// TIA Portal project "自动组装流水线（核心程序）" (V16)

(* hardware
DEVICE "S7-1200 station_1"  S7-1200 Station
   slot 0: "Rack_0"  S7-1200 Rack  Rack  V1.0
   slot 1: "PLC_1"  CPU 1214C DC/DC/Rly  6ES7 214-1HG40-0XB0  V4.4
*)

// ===== PLC "PLC_1"  CPU 1214C DC/DC/Rly =====

VAR_GLOBAL   // PLC tag table "io"
   "传感器9" AT %I0.0 : Bool;
   "传感器8" AT %I0.1 : Bool;
   "传感器7" AT %I0.2 : Bool;
   "传感器1" AT %I0.3 : Bool;
   "传感器2" AT %I0.4 : Bool;
   "传感器3" AT %I0.5 : Bool;
   "传感器4" AT %I0.6 : Bool;
   "传感器5" AT %I0.7 : Bool;
   "传感器6" AT %I1.0 : Bool;
   "传感器10" AT %I1.1 : Bool;
   "开始" AT %I1.2 : Bool;
   "复位" AT %I1.3 : Bool;
   "停止" AT %I1.4 : Bool;
   "紧急停止" AT %I1.5 : Bool;
   "1挡" AT %I1.6 : Bool;
   "FACTORY I/O (Running)" AT %I1.7 : Bool;
   "前后" AT %Q0.0 : Bool;
   "上下" AT %Q0.1 : Bool;
   "吸取" AT %Q0.2 : Bool;
   "皮带1" AT %Q0.3 : Bool;
   "推上盖" AT %Q0.4 : Bool;
   "上升1" AT %Q0.5 : Bool;
   "皮带2" AT %Q0.6 : Bool;
   "推下盖" AT %Q0.7 : Bool;
   "上升2" AT %Q1.0 : Bool;
   "绿灯" AT %Q1.1 : Bool;
   "黄灯" AT %Q1.2 : Bool;
   "红灯" AT %Q1.3 : Bool;
   "显示屏" AT %QD30 : DInt;
END_VAR

VAR_GLOBAL   // PLC tag table "中间变量"
   "中间变量1" AT %M0.0 : Bool;
   "中间变量2" AT %M0.1 : Bool;
   "中间变量3" AT %M0.2 : Bool;
   "中间变量4" AT %M0.3 : Bool;
   "中间变量5" AT %M0.4 : Bool;
   "中间变量6" AT %M0.5 : Bool;
   "中间变量7" AT %M0.6 : Bool;
   "中间变量8" AT %M0.7 : Bool;
   "中间变量9" AT %M1.0 : Bool;
   "中间变量10" AT %M1.1 : Bool;
   "中间变量11" AT %M1.2 : Bool;
   "中间变量12" AT %M1.3 : Bool;
   "中间变量13" AT %M1.4 : Bool;
   "中间变量14" AT %M1.5 : Bool;
   "启动" AT %M1.6 : Bool;
   "停止(1)" AT %M1.7 : Bool;
   "复位(1)" AT %M2.0 : Bool;
   "启动标志1" AT %M2.1 : Bool;
   "推杆标志1" AT %M2.2 : Bool;
   "推杆标志2" AT %M2.3 : Bool;
   "推杆收1" AT %M2.4 : Bool;
   "推杆收2" AT %M2.5 : Bool;
   "上下准备" AT %M2.6 : Bool;
   "吸附准备" AT %M2.7 : Bool;
   "吸附过程" AT %M3.0 : Bool;
   "前后准备" AT %M3.1 : Bool;
   "准备下降" AT %M3.2 : Bool;
   "断开吸附" AT %M3.3 : Bool;
   "x轴复位" AT %M3.4 : Bool;
   "皮带1状态" AT %M3.5 : Bool;
   "皮带2状态" AT %M3.6 : Bool;
   "皮带启动1" AT %M3.7 : Bool;
   "皮带启动2" AT %M4.0 : Bool;
   "上升2准备" AT %M4.1 : Bool;
   "上升2复位" AT %M4.2 : Bool;
END_VAR

// folder: System blocks/Program resources

DATA_BLOCK "IEC_Timer_0_DB"   // DB1
{ S7_Optimized_Access := 'TRUE' }
AUTHOR : Simatic
FAMILY : IEC
NAME : IEC_TMR
VERSION : 1.0
// stored: InstanceOfName IEC_TIMER
"IEC_TIMER"
BEGIN
END_DATA_BLOCK

DATA_BLOCK "IEC_Timer_0_DB_1"   // DB2
{ S7_Optimized_Access := 'TRUE' }
AUTHOR : Simatic
FAMILY : IEC
NAME : IEC_TMR
VERSION : 1.0
// stored: InstanceOfName IEC_TIMER
"IEC_TIMER"
BEGIN
END_DATA_BLOCK

DATA_BLOCK "IEC_Timer_0_DB_2"   // DB3
{ S7_Optimized_Access := 'TRUE' }
AUTHOR : Simatic
FAMILY : IEC
NAME : IEC_TMR
VERSION : 1.0
// stored: InstanceOfName IEC_TIMER
"IEC_TIMER"
BEGIN
END_DATA_BLOCK

DATA_BLOCK "IEC_Timer_0_DB_3"   // DB4
{ S7_Optimized_Access := 'TRUE' }
AUTHOR : Simatic
FAMILY : IEC
NAME : IEC_TMR
VERSION : 1.0
// stored: InstanceOfName IEC_TIMER
"IEC_TIMER"
BEGIN
END_DATA_BLOCK

DATA_BLOCK "IEC_Timer_0_DB_4"   // DB5
{ S7_Optimized_Access := 'TRUE' }
AUTHOR : Simatic
FAMILY : IEC
NAME : IEC_TMR
VERSION : 1.0
// stored: InstanceOfName IEC_TIMER
"IEC_TIMER"
BEGIN
END_DATA_BLOCK

DATA_BLOCK "IEC_Timer_0_DB_5"   // DB6
{ S7_Optimized_Access := 'TRUE' }
AUTHOR : Simatic
FAMILY : IEC
NAME : IEC_TMR
VERSION : 1.0
// stored: InstanceOfName IEC_TIMER
"IEC_TIMER"
BEGIN
END_DATA_BLOCK

DATA_BLOCK "IEC_Timer_0_DB_6"   // DB7
{ S7_Optimized_Access := 'TRUE' }
AUTHOR : Simatic
FAMILY : IEC
NAME : IEC_TMR
VERSION : 1.0
// stored: InstanceOfName IEC_TIMER
"IEC_TIMER"
BEGIN
END_DATA_BLOCK

DATA_BLOCK "IEC_Timer_0_DB_7"   // DB8
{ S7_Optimized_Access := 'TRUE' }
AUTHOR : Simatic
FAMILY : IEC
NAME : IEC_TMR
VERSION : 1.0
// stored: InstanceOfName IEC_TIMER
"IEC_TIMER"
BEGIN
END_DATA_BLOCK

DATA_BLOCK "IEC_Timer_0_DB_8"   // DB9
{ S7_Optimized_Access := 'TRUE' }
AUTHOR : Simatic
FAMILY : IEC
NAME : IEC_TMR
VERSION : 1.0
// stored: InstanceOfName IEC_TIMER
"IEC_TIMER"
BEGIN
END_DATA_BLOCK

DATA_BLOCK "IEC_Timer_0_DB_9"   // DB10
{ S7_Optimized_Access := 'TRUE' }
AUTHOR : Simatic
FAMILY : IEC
NAME : IEC_TMR
VERSION : 1.0
// stored: InstanceOfName IEC_TIMER
"IEC_TIMER"
BEGIN
END_DATA_BLOCK

DATA_BLOCK "IEC_Timer_0_DB_10"   // DB11
{ S7_Optimized_Access := 'TRUE' }
AUTHOR : Simatic
FAMILY : IEC
NAME : IEC_TMR
VERSION : 1.0
// stored: InstanceOfName IEC_TIMER
"IEC_TIMER"
BEGIN
END_DATA_BLOCK

DATA_BLOCK "IEC_Timer_0_DB_11"   // DB12
{ S7_Optimized_Access := 'TRUE' }
AUTHOR : Simatic
FAMILY : IEC
NAME : IEC_TMR
VERSION : 1.0
// stored: InstanceOfName IEC_TIMER
"IEC_TIMER"
BEGIN
END_DATA_BLOCK

// folder: (top level)

FUNCTION "MHJ-PLC-Lab-Function-S71200" : Void   // FC9000, SCL
{ S7_Optimized_Access := 'TRUE' }
VERSION : 0.1
   VAR_TEMP
      rdTimeReturn : Int;
      outputTime : DTL;
      SyncVal : Byte;
      forVal : Int;
      forVal_2 : Int;
      Value : Byte;
   END_VAR
   VAR CONSTANT
      CompVal : Byte := 16#34;
      Value_01 : Byte := 16#11;
      Value_01_DW : DWord := 16#A165_D992;
      Value_02_DW : DWord := 16#58BE_4401;
   END_VAR
BEGIN

   #Value:=PEEK(area := 16#82,
        dbNumber := 0,
        byteOffset := 511);
   #Value := #Value + 1;

   POKE(area := 16#82,
        dbNumber := 0,
        byteOffset := 511,
        value := #Value);

   POKE(area:=16#81,
        dbNumber:=0,
        byteOffset:=1016,
        value:=#Value_01_DW);
   POKE(area := 16#81,
        dbNumber := 0,
        byteOffset := 1020,
        value := #Value_02_DW);

   POKE(area := 16#81,
        dbNumber := 0,
        byteOffset := 511,
        value := B#16#00);

   FOR #forVal := 0 TO 120 DO
       FOR #forVal_2:=0 TO 10 DO
           #rdTimeReturn:=RD_SYS_T(#outputTime);
           #rdTimeReturn := WR_SYS_T(#outputTime);
           #rdTimeReturn := RD_SYS_T(#outputTime);
           #rdTimeReturn := WR_SYS_T(#outputTime);
       END_FOR;
       #SyncVal:= PEEK(area := 16#81,
                      dbNumber := 0,
                      byteOffset := 511);
       IF #SyncVal = #CompVal THEN
          GOTO M_1;
       END_IF;
   END_FOR;
   RETURN;

   M_1:
   POKE(area := 16#81,
        dbNumber := 0,
        byteOffset := 511,
        value := B#16#0);
END_FUNCTION

ORGANIZATION_BLOCK "Main"   // OB1, LAD, ProgramCycle
TITLE = "Main Program Sweep (Cycle)"
{ S7_Optimized_Access := 'TRUE' }
VERSION : 0.1
   VAR_INPUT
      Initial_Call : Bool;   // Initial call of this OB
      Remanence : Bool;   // =True, if remanent data are available
   END_VAR
   VAR_TEMP   // added for the SCL form of the ladder/FBD networks
      _w1 : Bool;
      _w2 : Bool;
   END_VAR
BEGIN

REGION Network 1
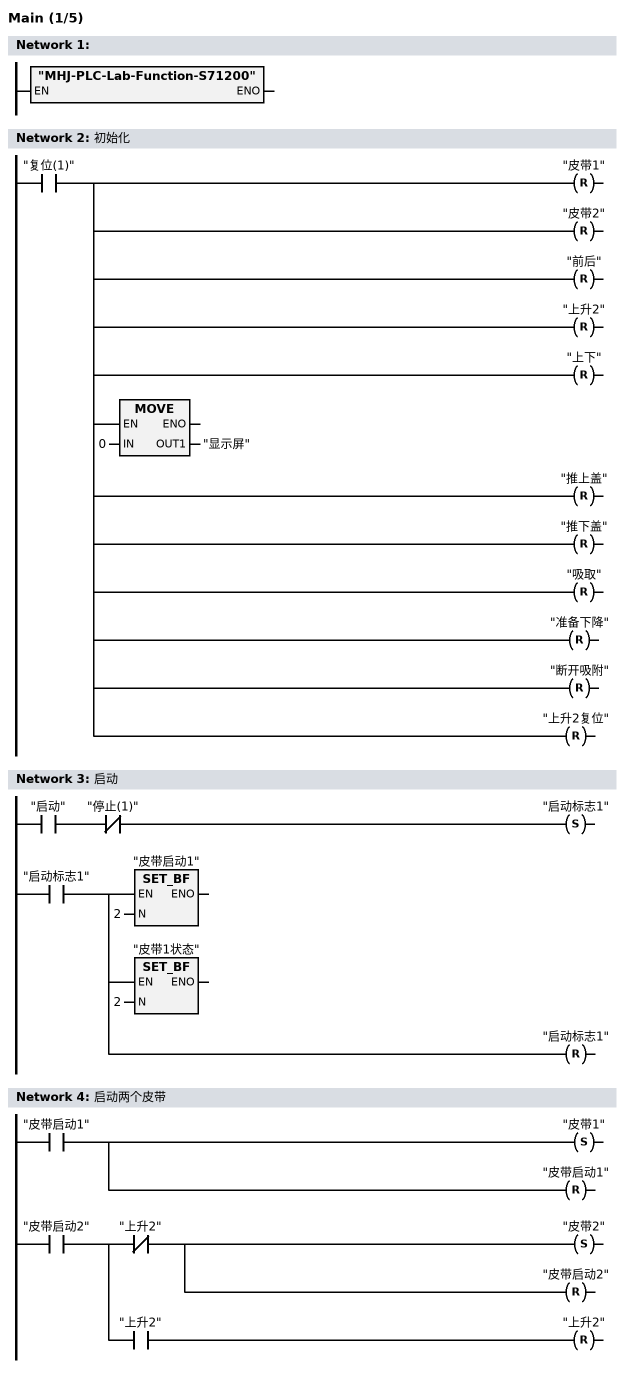
   RUNG wire#powerrail
      "MHJ-PLC-Lab-Function-S71200"()
   END_RUNG
   // the same network as SCL:
   "MHJ-PLC-Lab-Function-S71200"();
END_REGION

REGION Network 2: 初始化
   RUNG wire#powerrail
      Contact( "复位(1)" )
      wire#w1
      R_Coil( "皮带1" )
   END_RUNG
   RUNG wire#w1
      R_Coil( "皮带2" )
   END_RUNG
   RUNG wire#w1
      R_Coil( "前后" )
   END_RUNG
   RUNG wire#w1
      R_Coil( "上升2" )
   END_RUNG
   RUNG wire#w1
      R_Coil( "上下" )
   END_RUNG
   RUNG wire#w1
      Move(in := 0, out1 => "显示屏")
   END_RUNG
   RUNG wire#w1
      R_Coil( "推上盖" )
   END_RUNG
   RUNG wire#w1
      R_Coil( "推下盖" )
   END_RUNG
   RUNG wire#w1
      R_Coil( "吸取" )
   END_RUNG
   RUNG wire#w1
      R_Coil( "准备下降" )
   END_RUNG
   RUNG wire#w1
      R_Coil( "断开吸附" )
   END_RUNG
   RUNG wire#w1
      R_Coil( "上升2复位" )
   END_RUNG
   // the same network as SCL:
   IF "复位(1)" THEN
       "皮带1" := FALSE;
       "皮带2" := FALSE;
       "前后" := FALSE;
       "上升2" := FALSE;
       "上下" := FALSE;
       "显示屏" := 0;
       "推上盖" := FALSE;
       "推下盖" := FALSE;
       "吸取" := FALSE;
       "准备下降" := FALSE;
       "断开吸附" := FALSE;
       "上升2复位" := FALSE;
   END_IF;
END_REGION

REGION Network 3: 启动
   // no SCL statement known for SBitfield: written as a call
   IF "启动" AND NOT "停止(1)" THEN "启动标志1" := TRUE; END_IF;
   #_w1 := "启动标志1";
   IF #_w1 THEN
       SET_BF(operand := "皮带启动1", n := 2);
       SET_BF(operand := "皮带1状态", n := 2);
       "启动标志1" := FALSE;
   END_IF;
END_REGION

REGION Network 4: 启动两个皮带
   RUNG wire#powerrail
      Contact( "皮带启动1" )
      wire#w1
      S_Coil( "皮带1" )
   END_RUNG
   RUNG wire#w1
      R_Coil( "皮带启动1" )
   END_RUNG
   RUNG wire#powerrail
      Contact( "皮带启动2" )
      wire#w2
      I_Contact( "上升2" )
      wire#w3
      S_Coil( "皮带2" )
   END_RUNG
   RUNG wire#w3
      R_Coil( "皮带启动2" )
   END_RUNG
   RUNG wire#w2
      Contact( "上升2" )
      R_Coil( "上升2" )
   END_RUNG
   // the same network as SCL:
   IF "皮带启动1" THEN
       "皮带1" := TRUE;
       "皮带启动1" := FALSE;
   END_IF;
   IF "皮带启动2" AND NOT "上升2" THEN "皮带2" := TRUE; END_IF;
   #_w1 := "皮带启动2";
   IF "皮带启动2" AND NOT "上升2" THEN "皮带启动2" := FALSE; END_IF;
   IF #_w1 AND "上升2" THEN "上升2" := FALSE; END_IF;
END_REGION

REGION Network 5: 停止传送带运动，启动两个推杆
   // 因为传感器从1变为0在显示上面有延迟的存在，在电脑内部的运行中没有，所以需要延时一段时间，再停止运行皮带，开始运行推杆
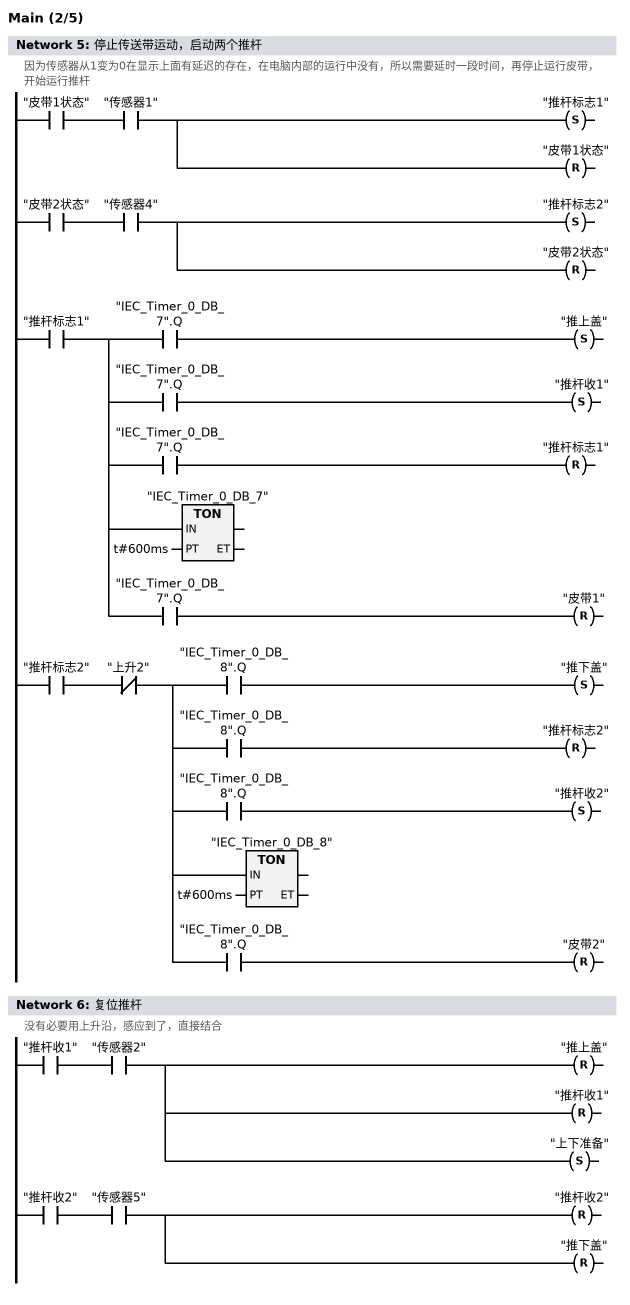
   IF "皮带1状态" AND "传感器1" THEN
       "推杆标志1" := TRUE;
       "皮带1状态" := FALSE;
   END_IF;
   IF "皮带2状态" AND "传感器4" THEN
       "推杆标志2" := TRUE;
       "皮带2状态" := FALSE;
   END_IF;
   IF "推杆标志1" AND "IEC_Timer_0_DB_7".Q THEN
       "推上盖" := TRUE;
       "推杆收1" := TRUE;
   END_IF;
   #_w1 := "推杆标志1";
   IF "推杆标志1" AND "IEC_Timer_0_DB_7".Q THEN "推杆标志1" := FALSE; END_IF;
   "IEC_Timer_0_DB_7".TON(IN := #_w1, PT := t#600ms);
   IF #_w1 AND "IEC_Timer_0_DB_7".Q THEN "皮带1" := FALSE; END_IF;
   #_w2 := "推杆标志2" AND NOT "上升2";
   IF #_w2 AND "IEC_Timer_0_DB_8".Q THEN
       "推下盖" := TRUE;
       "推杆标志2" := FALSE;
       "推杆收2" := TRUE;
   END_IF;
   "IEC_Timer_0_DB_8".TON(IN := #_w2, PT := t#600ms);
   IF #_w2 AND "IEC_Timer_0_DB_8".Q THEN "皮带2" := FALSE; END_IF;
END_REGION

REGION Network 6: 复位推杆
   // 没有必要用上升沿，感应到了，直接结合
   RUNG wire#powerrail
      Contact( "推杆收1" )
      Contact( "传感器2" )
      wire#w1
      R_Coil( "推上盖" )
   END_RUNG
   RUNG wire#w1
      R_Coil( "推杆收1" )
   END_RUNG
   RUNG wire#w1
      S_Coil( "上下准备" )
   END_RUNG
   RUNG wire#powerrail
      Contact( "推杆收2" )
      Contact( "传感器5" )
      wire#w2
      R_Coil( "推杆收2" )
   END_RUNG
   RUNG wire#w2
      R_Coil( "推下盖" )
   END_RUNG
   // the same network as SCL:
   IF "推杆收1" AND "传感器2" THEN "推上盖" := FALSE; END_IF;
   #_w1 := "推杆收1" AND "传感器2";
   IF #_w1 THEN
       "推杆收1" := FALSE;
       "上下准备" := TRUE;
   END_IF;
   #_w2 := "推杆收2" AND "传感器5";
   IF #_w2 THEN
       "推杆收2" := FALSE;
       "推下盖" := FALSE;
   END_IF;
END_REGION

REGION Network 7: 准备吸附
   // 利用传感器2来判断是否推到位
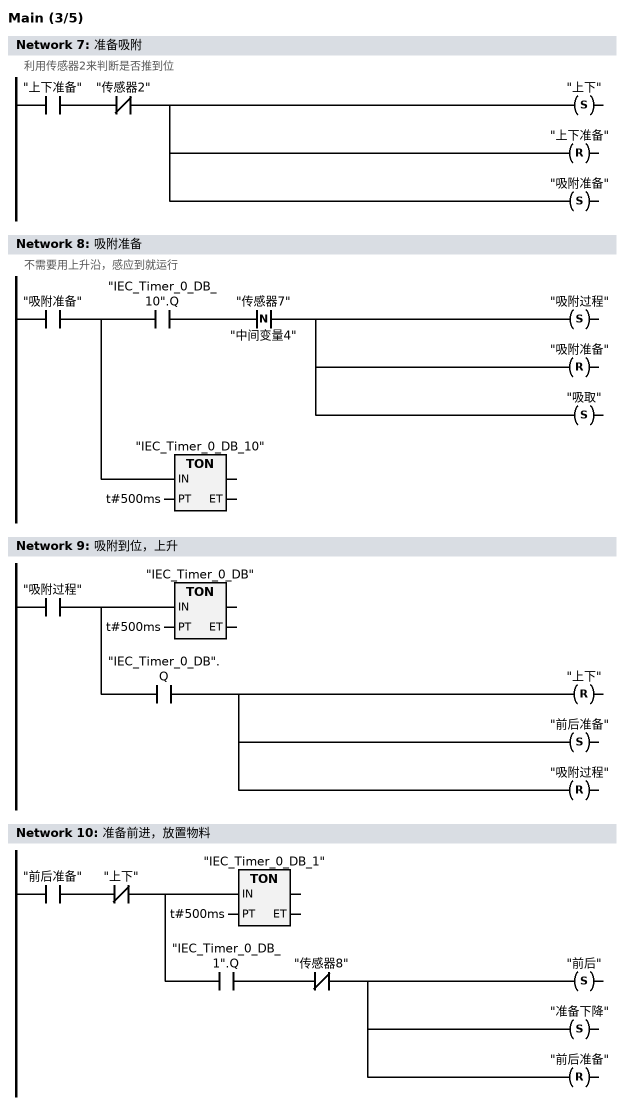
   RUNG wire#powerrail
      Contact( "上下准备" )
      I_Contact( "传感器2" )
      wire#w1
      S_Coil( "上下" )
   END_RUNG
   RUNG wire#w1
      R_Coil( "上下准备" )
   END_RUNG
   RUNG wire#w1
      S_Coil( "吸附准备" )
   END_RUNG
   // the same network as SCL:
   IF "上下准备" AND NOT "传感器2" THEN "上下" := TRUE; END_IF;
   #_w1 := "上下准备" AND NOT "传感器2";
   IF #_w1 THEN
       "上下准备" := FALSE;
       "吸附准备" := TRUE;
   END_IF;
END_REGION

REGION Network 8: 吸附准备
   // 不需要用上升沿，感应到就运行
   #_w1 := "吸附准备" AND "IEC_Timer_0_DB_10".Q AND NOT "传感器7" AND "中间变量4";   // falling edge of "传感器7"
   "中间变量4" := "传感器7";
   IF #_w1 THEN "吸附过程" := TRUE; END_IF;
   #_w2 := "吸附准备";
   IF #_w1 THEN
       "吸附准备" := FALSE;
       "吸取" := TRUE;
   END_IF;
   "IEC_Timer_0_DB_10".TON(IN := #_w2, PT := t#500ms);
END_REGION

REGION Network 9: 吸附到位，上升
   "IEC_Timer_0_DB".TON(IN := "吸附过程", PT := t#500ms);
   IF "吸附过程" AND "IEC_Timer_0_DB".Q THEN
       "上下" := FALSE;
       "前后准备" := TRUE;
       "吸附过程" := FALSE;
   END_IF;
END_REGION

REGION Network 10: 准备前进，放置物料
   #_w1 := "前后准备" AND NOT "上下";
   "IEC_Timer_0_DB_1".TON(IN := #_w1, PT := t#500ms);
   IF #_w1 AND "IEC_Timer_0_DB_1".Q AND NOT "传感器8" THEN
       "前后" := TRUE;
       "准备下降" := TRUE;
       "前后准备" := FALSE;
   END_IF;
END_REGION

REGION Network 11
   // 利用传感器不运动的时候，表示为0
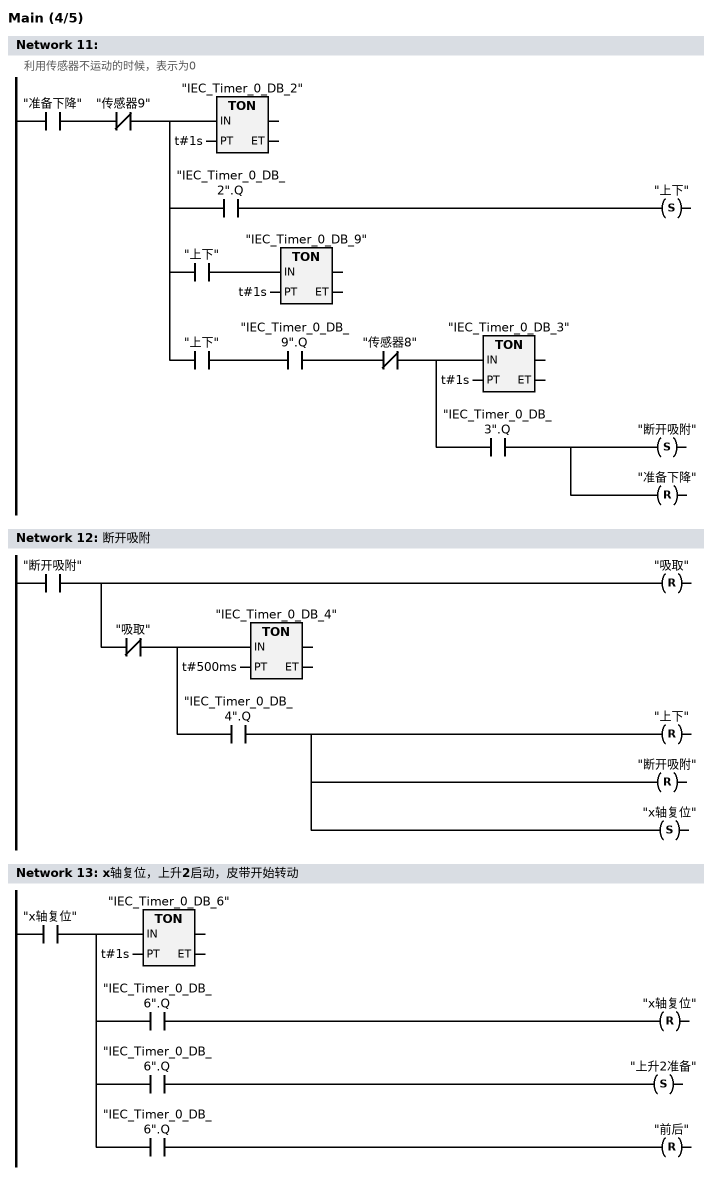
   #_w1 := "准备下降" AND NOT "传感器9";
   "IEC_Timer_0_DB_2".TON(IN := #_w1, PT := t#1s);
   IF #_w1 AND "IEC_Timer_0_DB_2".Q THEN "上下" := TRUE; END_IF;
   "IEC_Timer_0_DB_9".TON(IN := #_w1 AND "上下", PT := t#1s);
   #_w2 := #_w1 AND "上下" AND "IEC_Timer_0_DB_9".Q AND NOT "传感器8";
   "IEC_Timer_0_DB_3".TON(IN := #_w2, PT := t#1s);
   IF #_w2 AND "IEC_Timer_0_DB_3".Q THEN
       "断开吸附" := TRUE;
       "准备下降" := FALSE;
   END_IF;
END_REGION

REGION Network 12: 断开吸附
   IF "断开吸附" THEN "吸取" := FALSE; END_IF;
   #_w1 := "断开吸附" AND NOT "吸取";
   "IEC_Timer_0_DB_4".TON(IN := #_w1, PT := t#500ms);
   IF #_w1 AND "IEC_Timer_0_DB_4".Q THEN
       "上下" := FALSE;
       "断开吸附" := FALSE;
       "x轴复位" := TRUE;
   END_IF;
END_REGION

REGION Network 13: x轴复位，上升2启动，皮带开始转动
   "IEC_Timer_0_DB_6".TON(IN := "x轴复位", PT := t#1s);
   #_w1 := "x轴复位";
   IF "x轴复位" AND "IEC_Timer_0_DB_6".Q THEN "x轴复位" := FALSE; END_IF;
   IF #_w1 AND "IEC_Timer_0_DB_6".Q THEN
       "上升2准备" := TRUE;
       "前后" := FALSE;
   END_IF;
END_REGION

REGION Network 14: 准备循环
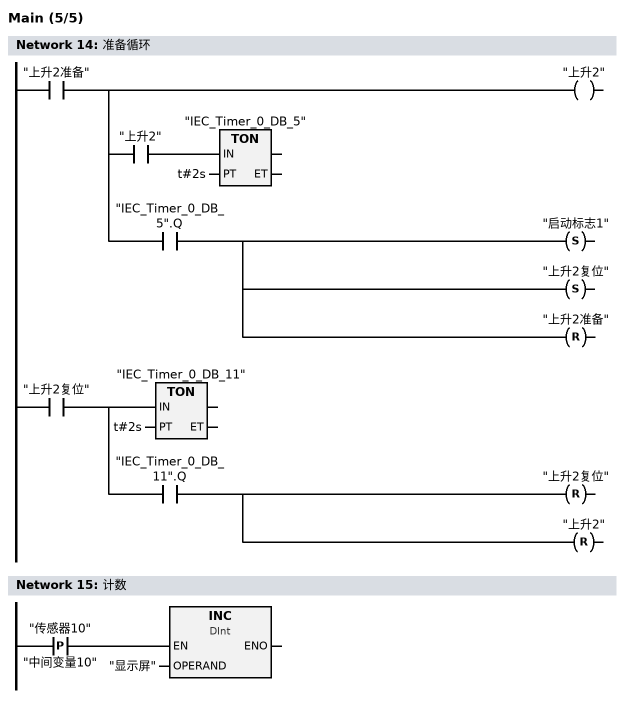
   "上升2" := "上升2准备";
   "IEC_Timer_0_DB_5".TON(IN := "上升2准备" AND "上升2", PT := t#2s);
   IF "上升2准备" AND "IEC_Timer_0_DB_5".Q THEN
       "启动标志1" := TRUE;
       "上升2复位" := TRUE;
       "上升2准备" := FALSE;
   END_IF;
   "IEC_Timer_0_DB_11".TON(IN := "上升2复位", PT := t#2s);
   #_w1 := "上升2复位" AND "IEC_Timer_0_DB_11".Q;
   IF #_w1 THEN
       "上升2复位" := FALSE;
       "上升2" := FALSE;
   END_IF;
END_REGION

REGION Network 15: 计数
   RUNG wire#powerrail
      P_Contact(operand := "传感器10", bit := "中间变量10")
      { S7_Templates := "DestType := DInt" } Inc( "显示屏" )
   END_RUNG
   // the same network as SCL:
   #_w1 := "传感器10" AND NOT "中间变量10";   // rising edge of "传感器10"
   "中间变量10" := "传感器10";
   IF #_w1 THEN "显示屏" := "显示屏" + 1; END_IF;
END_REGION
END_ORGANIZATION_BLOCK